INTERFACE I_CommandTask EXTENDS I_Task

METHOD PUBLIC Initalise : BOOL
VAR_INPUT
 comPort : I_Connection;
 msg : T_Maxstring;
END_VAR
END_METHOD

END_INTERFACE

(* stored: Version 1.1.0.1
   Itf I_CommandTask: Id {ee4d4c1e-f281-4297-99e2-d750d653835a}
   Folder Methods: Id {43c92586-db72-423c-9ec8-8ac578a6d493}
   Method Initalise: Id {e6fb384a-3d96-40ec-b318-8af562015284} *)
